Staubli VAL3: sampleChangerv5.pjx

--- sampleChangerv5.pjx ---
Parameters version=s7.7 stackSize=5000 millimeterUnit=true
Program file=comm.pgx
Program file=getNearestPos.pgx
Program file=getPosition.pgx
Program file=moveManager.pgx
Program file=observeStop.pgx
Program file=powerSwitch.pgx
Program file=sampleGripping.pgx
Program file=sendStatus.pgx
Program file=setSamPosOffs.pgx
Program file=setSpeed.pgx
Program file=setSpinPosOffs.pgx
Program file=start.pgx
Program file=stop.pgx
Program file=test.pgx
Program file=zsetSpinPosOffs.pgx
Data file=sampleChangerv5.dtx

--- sampleChangerV4.dtx ---
bool taskIsDone
dio switchGripper = {link=valve1}
jointRx binPosition = {j1=59.154914, j2=15.287075, j3=144.068937, j4=0.00349, j5=20.640131, j6=239.148927}
jointRx currentPickPosJ = {j1=24.086468, j2=103.725715, j3=36.339858, j4=-71.090092, j5=105.162663, j6=322.602811}
jointRx currentSamPosJ = {j1=64.5166, j2=21.7725, j3=135.395, j4=0.005, j5=22.8226, j6=244.506}
jointRx gatePosition = {j1=53.332436, j2=31.008098, j3=108.023775, j4=-0.035914, j5=40.963114, j6=323.353672}
jointRx homePosition = {j1=64.5166, j2=21.7725, j3=135.395, j4=0.005, j5=22.8226, j6=244.506}
jointRx parkingPosition = {j1=20.774519, j2=86.925335, j3=58.285959, j4=-72.455135, j5=101.349332, j6=295.989419}
jointRx spinnerPosition = {j1=24.224814, j2=103.543996, j3=36.557875, j4=-70.964584, j5=105.220885, j6=322.664695}
jointRx zeroPosition = {j1=88.745927, j2=-26.51301, j3=117.695598, j4=-0.539561, j5=89.308877, j6=269.442332}
mdesc mFastMov = {blend=off}
mdesc mNomSpeed = {accel=2.25, vel=15, decel=2.25}
num coords[2]
  [0] = 4
  [1] = 9
num numMessage[32]
num numSpeed = 5
num numXarray = 1
num numXold
num numYarray = 1
num numYold
pointRx currentPickPos = {x=982.652852, y=394.034002, z=-652.657917, rx=90.013165, ry=0.023145, rz=89.994895, shoulder=lefty, elbow=epositive, wrist=wpositive, fatherId=world[0]}
pointRx currentSamPos = {x=188.431145, y=511.898865, z=-95.729646, rx=-179.992666, ry=0.001448, rz=-0.004557, shoulder=lefty, elbow=epositive, wrist=wpositive, fatherId=world[0]}
sio sioASCII[2]
  [0] = {link=Socket\tan}
  [1] = {link=Socket\tan}

--- sampleChangerv5.dtx ---
bool moveIsStopped
dio switchGripper = {link=valve1}
jointRx binPosition = {j1=59.154914, j2=15.287075, j3=144.068937, j4=0.00349, j5=20.640131, j6=239.148927}
jointRx currentSamPosJ = {j1=64.5166, j2=21.7725, j3=135.395, j4=0.005, j5=22.8226, j6=244.506}
jointRx currentSpinPosJ
jointRx gatePosition = {j1=53.332436, j2=31.008098, j3=108.023775, j4=-0.035914, j5=40.963114, j6=323.353672}
jointRx homePosition = {j1=64.5166, j2=21.7725, j3=135.395, j4=0.005, j5=22.8226, j6=244.506}
jointRx knownPositions{}
  [currentSamPos] = {}
  [currentSpinPos] = {}
  [gatePosition] = {}
  [homePosition] = {}
  [parkingPosition] = {}
  [spinnerHomePos] = {}
  [zeroPosition] = {}
  [binPosition] = {}
jointRx parkingPosition = {j1=20.774519, j2=86.925335, j3=58.285959, j4=-72.455135, j5=101.349332, j6=295.989419}
jointRx spinnerHomePos = {j1=24.038951, j2=102.353577, j3=38.089715, j4=-71.031763, j5=105.005317, j6=322.961782}
jointRx zeroPosition = {j1=88.745927, j2=-26.51301, j3=117.695598, j4=-0.539561, j5=89.308877, j6=269.442332}
mdesc mFastMov = {blend=off}
mdesc mNomSpeed = {accel=2.25, vel=15, decel=2.25}
num numSamOffs[2]
num numSpinOffs[6]
sio sioASCII[2]
  [0] = {link=Socket\tan}
  [1] = {link=Socket\tan}
bool mounted
string calibInfo

--- start.pgx ---
program start()
begin
  call comm()
end

--- closeGripper.pgx ---
program closeGripper()
begin
  switchGripper=false
  taskKill("closeGripper")
end

--- comm.pgx ---
program comm()
  local num asciiMessage[64]
  local string command
  local string gripState
  local num nchars
  local string reply
  local num sio_ID
  local string stringMessage
  local num stringPos
  local bool waitForMessage
  local num msgLength
begin
  put("Starting sampleChangerV5.1...")
  //Disconnect running sessions
  clearBuffer(sioASCII)
  // We initialise the current sample position as the homePosition for safety's sake!
  currentSamPosJ=homePosition
  stringMessage=""
  reply=""
  msgLength=0

  // Populate the collection of known positions
  knownPositions["binPosition"] = binPosition
  knownPositions["currentSamPos"] = currentSamPosJ
  knownPositions["currentSpinPos"] = currentSpinPosJ
  knownPositions["gatePosition"] = gatePosition
  knownPositions["homePosition"] = homePosition
  knownPositions["parkingPosition"] = parkingPosition
  knownPositions["spinnerHomePos"] = spinnerHomePos
  knownPositions["zeroPosition"] = zeroPosition

  userPage()
  cls()

  putln("sampleChangerV5.1 server started.")
  putln("Waiting for command...")

  // Provides the server-like behaviour
  while true

    // The next while loop handles receiving messages.
    // The only way out is to recieve a message terminated with a ;
    waitForMessage=true
    while waitForMessage
      // The sioASCII socket allows two connections. We need to check which has something it it
      // Read recv buffer & place ASCII values in asciiMessage
      nchars=sioGet(sioASCII[0],asciiMessage)
      if nchars>0
        sio_ID=0
      else
        nchars=sioGet(sioASCII[1],asciiMessage)
        if nchars>0
          sio_ID=1
        else
        endIf
      endIf
      // Useful for debugging how many chars were received by the server
      //put("nchars: ")
      //putln(nchars)

      // sioGet returns a ASCII bytes. We need to decode them.
      if nchars>0
        stringMessage=chr(asciiMessage[0])
        for stringPos=1 to 63
          stringMessage=stringMessage+chr(asciiMessage[stringPos])
        endFor
        // We are finished with asciiMessage. Clear it
        for stringPos=0 to 63
          asciiMessage[stringPos]=0
        endFor

        // Check the last character in the message was a message end char (;)
        // If not, inform the sender and don't do anything
        if right(stringMessage,1)==";"
          stringMessage=left(stringMessage,len(stringMessage)-1)
          waitForMessage=false
        else
          call sendStatus(":fail_'No message end'",sio_ID)
          stringMessage=""
        endIf
        // Useful for debugging what was received by the server
        //put("stringMessage: ")
        //putln(stringMessage)
      endIf
    endWhile


    // All incoming messages should be of the form:
    //   command[:parameters]
    // Trim off the parameters for the switch statement
    stringPos=find(stringMessage,":")
    if stringPos>0
      command=left(stringMessage,stringPos)
    else
      command=stringMessage
    endIf
    put("Command: ")
    putln(command)

    //Now decide how to handle the message
    switch command
      // Testing routines
      // **********
      case "hello"
        call sendStatus("world",sio_ID)
      break

      case "test"
        call test()
      break

      // Control routines
      // **********
      case "setSamPosOffset"
        taskCreate "setSamPosOffset",10,setSamPosOffs(stringMessage,sio_ID)
        wait(taskStatus("setSamPosOffset")==-1)
      break

      case "getSamPosOffset"
        reply="getSamPosOffset:#X"+toString(".3",numSamOffs[0])
        reply=reply+"#Y"+toString(".3",numSamOffs[1])
        call sendStatus(reply,sio_ID)
      break

      case "setSpinPosOffset"
        taskCreate "setSpinPosOff",10,setSpinPosOffs(stringMessage,sio_ID)
        wait(taskStatus("setSpinPosOff")==-1)
      break

      case "getSpinPosOffset"
        reply="getSpinPosOffset:#X"+toString(".3",numSpinOffs[0])+"#Y"+toString(".3",numSpinOffs[1])
        reply=reply+"#Z"+toString(".3",numSpinOffs[2])+"#RX"+toString(".1",numSpinOffs[3])
        reply=reply+"#RY"+toString(".1",numSpinOffs[4])+"#RZ"+toString(".1",numSpinOffs[5])
        call sendStatus(reply,sio_ID)
      break

      case "getSpinPosition"
        call getPosition("getSpinPosition",currentSpinPosJ,sio_ID)
      break

      case "getSpinHomePosition"
        call getPosition("getSpinHomePosition",spinnerHomePos,sio_ID)
      break

      case "getCurrentPosition"
        call getPosition("getCurrentPosition",herej(),sio_ID)
      break

      case "getNearestPosition"
        call getNearestPos(sio_ID)
      break

      case "setCalibInfo"
        // Sets calibration info string
        msgLength = len(stringMessage)
        calibInfo = mid(stringMessage, (msgLength - 13), 13)
        call sendStatus("setCalibInfo:done", sio_ID)
      break

      case "getCalibInfo"
       reply = "getCalibInfo:" + calibInfo
       call sendStatus(reply,sio_ID)
      break

      case "setSpeed"
        taskCreate "setSpeed",5,setSpeed(stringMessage,sio_ID)
        wait(taskStatus("setSpeed")==-1)
      break

      case "getSpeed"
        call sendStatus("getSpeed:#"+toString("",mFastMov.vel),sio_ID)
      break

      case "powerOn"
        putln("Enabling robot power ...")
        taskCreate "powerSwitch",10,powerSwitch(true,"powerOn",sio_ID)
      break

      case "powerOff"
        putln("Disabling robot power ...")
        taskCreate "powerSwitch",10,powerSwitch(false,"powerOff",sio_ID)
      break

      case "getPowerState"
        putln("Get power status ...")
        if (isPowered()==false)
          reply="getPowerState:#Off"
        else
          reply="getPowerState:#On"
        endIf
        taskCreate "sendStatus",10,sendStatus(reply,sio_ID)
      break

      case "interrupt"
        putln("Interrupt movement ...")
        // Temporarily stops movement. This is basically a pause!\
        // Used by observeStop
        moveIsStopped=true
        call sendStatus("interrupt:done", sio_ID)
      break

      case "restart"
        putln("Restart from interruption ...")
        // Used by observeStop
        moveIsStopped=false
        call sendStatus("restart:done", sio_ID)
      break

      case "getGripperState"
        if switchGripper==true
          gripState="closed"
        else
          gripState="open"
        endIf
        call sendStatus("getGripperState:"+gripState,sio_ID)
      break

      // Movement routines
      // **********
      // Home position for the sample (sam)
      case "moveHome"
        putln("Moving to home ...")
        taskCreate "moveHome",10,moveManager(homePosition,mFastMov,"moveHome:done",sio_ID)
      break

      //Move to current sample offset position (home + offset)
      case "moveSamPos"
        putln("Moving to current sample ...")
        taskCreate "moveSamPos",10,moveManager(currentSamPosJ,mFastMov,"moveSamPos:done",sio_ID)
      break

      case "moveGate"
        putln("Moving to gate ...")
        taskCreate "moveGate",10,moveManager(gatePosition,mFastMov,"moveGate:done",sio_ID)
      break

      // Home position (calibrated) for the spinner
      case "moveSpinHome"
        putln("Moving to spinner home ...")
        taskCreate "moveSpinHome",10,moveManager(spinnerHomePos,mFastMov,"moveSpinHome:done",sio_ID)
      break

      //Move to current spinner offset position (spinnerHome + offset)
      case "moveSpinner"
        putln("Moving to spinner ...")
        taskCreate "moveSpinner",10,moveManager(currentSpinPosJ,mFastMov,"moveSpinner:done",sio_ID)
      break

      case "moveOffside"
        putln("Moving to offside ...")
        taskCreate "moveOffside",10,moveManager(parkingPosition,mFastMov,"moveOffside:done",sio_ID)
      break

      case "moveZero"
        putln("Moving to zero ...")
        taskCreate "moveZero",10,moveManager(zeroPosition,mFastMov,"moveZero:done",sio_ID)
      break

      case "moveBin"
        putln("Moving to bin ...")
        taskCreate "moveBin",10,moveManager(binPosition,mFastMov,"moveBin:done",sio_ID)
      break

      // Sample Handling
      // **********
      case "samplePick"
        putln("Picking sample ...")
        taskCreate "sampleGripping",10,sampleGripping(true,"samplePick",sio_ID)
      break

      case "sampleRelease"
        putln("Releasing sample ...")
        taskCreate "sampleGripping",10,sampleGripping(false,"sampleRelease",sio_ID)
      break

      case "gripperOpen"
        putln("Open gripper ...")
        switchGripper=false
        taskCreate "sendStatus",10,sendStatus("gripperOpen:done",sio_ID)
      break

      case "gripperClose"
        putln("Close gripper ...")
        switchGripper=true
        taskCreate "sendStatus",10,sendStatus("gripperClose:done",sio_ID)
      break

      case "isSampleMounted"
        // Check the state of the sample mounted flag
        if mounted == true
          reply = "isSampleMounted:#Yes"
        else
          reply = "isSampleMounted:#No"
        endIf
        call sendStatus(reply, sio_ID)
      break

      case "sampleMounted"
        // Set the sample mounted flag mounted (this is only s software flag)
        mounted = true
        taskCreate "sendStatus", 10, sendStatus("sampleMounted:done", sio_ID)
      break

      case "sampleUnmounted"
        // Set the sample mounted flag not mounted (this is only a software flag)
        mounted = false
        taskCreate "sendStatus", 10, sendStatus("sampleUnmounted:done", sio_ID)
      break

      default
        call sendStatus(":fail_'Unrecognised Command!'",sio_ID)
      break

    endSwitch
    // This message has been processed, so clear the stringMessage/command
    stringMessage=""
    command=""
    sio_ID=-1
    reply=""
    msgLength=0

  endWhile
end

--- getPosition.pgx ---
program getPosition(string getCommandName, joint requestedJoint, num sio_ID)
  local string message
  local pointRx readPosition
begin
  //**************************************************
  // Returns the contents of the trsf of the requested position.
  // On testing, we found that whereas a distance can be requested with
  // 2 or 3dp of precision, angles could not (got a runtime error on
  // the robot. Hence we return angles with no dp; we only need 2dp for
  // distances.
  //**************************************************
  putln("getPosition:")
  putln("   "+getCommandName)
  readPosition=jointToPoint(flange,world,requestedJoint)
  message=getCommandName+":#X"+toString(".2",readPosition.trsf.x)
  message=message+"#Y"+toString(".2",readPosition.trsf.y)
  message=message+"#Z"+toString(".2",readPosition.trsf.z)
  message=message+"#RX"+toString("",readPosition.trsf.rx)
  message=message+"#RY"+toString("",readPosition.trsf.ry)
  message=message+"#RZ"+toString("",readPosition.trsf.rz)

  call sendStatus(message,sio_ID)
end

--- moveBin.pgx ---
program moveBin()
begin
  movej(binPosition,flange,mFastMov)
  waitEndMove()
  message="moveBin:done"
  taskCreate "sendStatus",10,sendStatus()
  taskKill("moveBin")
end

--- moveGate.pgx ---
program moveGate()
begin
  movej(gatePosition,flange,mFastMov)
  waitEndMove()
  message="moveGate:done"
  taskCreate "sendStatus",100,sendStatus()
  taskKill("moveGate")
end

--- moveHome.pgx ---
program moveHome()
begin
  movej(homePosition,flange,mFastMov)
  waitEndMove()
  message="moveHome:done"
  taskCreate "sendStatus",100,sendStatus()
  taskKill("moveHome")
end

--- moveManager.pgx ---
program moveManager(joint destination (dimensions=1), mdesc armSpeed (dimensions=1), string reply (dimensions=1), num sio_ID (dimensions=1))
begin
  //**************************************************
  // Method to enable joint-based movements of the robot. The referenced
  // observeStop() method allows interrupts/restarts to be handled
  //**************************************************
  taskIsDone=false
  taskCreate "observeStop",5,observeStop()
  movej(destination,flange,armSpeed)
  waitEndMove()
  taskCreate "sendStatus",10,sendStatus(reply,sio_ID)
  taskKill("observeStop")
end

--- moveNext.pgx ---
program moveNext()
begin
  currentSamPosJ=herej()
  currentSamPos=jointToPoint(flange,world,currentSamPosJ)
  movel(appro(currentSamPos,{(numXarray-1)*-17.03,(numYarray-1)*-17,0,0,0,0}),flange,mFastMov)
  waitEndMove()
end

--- moveOffside.pgx ---
program moveOffside()
begin
  movej(parkingPosition,flange,mFastMov)
  waitEndMove()
  message="moveOffside:done"
  taskCreate "sendStatus",100,sendStatus()
  taskKill("moveOffside")
end

--- moveSpinner.pgx ---
program moveSpinner()
begin
  movej(spinnerPosition,flange,mFastMov)
  waitEndMove()
  message="moveSpinner:done"
  taskCreate "sendStatus",100,sendStatus()
  taskKill("moveSpinner")
end

--- moveZero.pgx ---
program moveZero()
begin
  movej(zeroPosition,flange,mFastMov)
  waitEndMove()
  message="moveZero:done"
  taskCreate "sendStatus",100,sendStatus()
  taskKill("moveZero")
end

--- notGrip.pgx ---
program notGrip()
begin
  if switchGripper==true
    switchGripper=false
  else
  endIf
end

--- observeStop.pgx ---
program observeStop()
begin
  //**************************************************
  // Method interrupts a running move operation. This is
  // equivalent to a pause.
  //
  // Method is triggered by a flag being set.
  // N.B. Move is only stopped until flag is unset.
  //**************************************************
  while true
    wait(moveIsStopped==true)
    stopMove()
    wait(moveIsStopped==false)
    restartMove()
  endWhile
end

--- openGripper.pgx ---
program openGripper()
begin
  switchGripper=false
  message="openGripper:done"
  taskCreate "sendStatus",100,sendStatus()
  taskKill("openGripper")
end

--- pickSample.pgx ---
program pickSample()
begin
  taskCreate "notGrip",100,notGrip()
  currentSamPosJ=herej()
  currentSamPos=jointToPoint(flange,world,currentSamPosJ)
  movel(appro(currentSamPos,{0,0,80,0,0,0}),flange,mNomSpeed)
  waitEndMove()
  taskKill("notGrip")
  switchGripper=true
  movel(appro(currentSamPos,{0,0,0,0,0,0}),flange,mNomSpeed)
  waitEndMove()
  message="pickSample:done"
  taskCreate "sendStatus",100,sendStatus()
  taskKill("pickSample")
  //taskKill("notGrip")
end

--- powerOff.pgx ---
program powerOff()
begin
  disablePower()
  message="disablePower:done"
  taskCreate "sendStatus",100,sendStatus()
  taskKill ("powerOff")
end

--- powerOn.pgx ---
program powerOn()
begin
 enablePower()
 if (watch(isPowered(),5)==false)
  putln("Arm power supply cannot be switched on")
 endIf
 message="enablePower:done"
 taskCreate "sendStatus",100,sendStatus()
 taskKill ("powerOn")
end

--- powerSwitch.pgx ---
program powerSwitch(bool enable (dimensions=1), string command (dimensions=1), num sio_ID (dimensions=1))
  local string reply
begin
  //**************************************************
  // Method to enable or disable the power on the robot, depending whether the
  // enable variable is true or false. Command argument is needed to construct
  // the reply
  //**************************************************
  if enable
    enablePower()
  else
    disablePower()
  endIf

  if (watch(isPowered()==enable,5)==false)
    reply=command+":fail_'RobotPowerCannotBeSwitched'"
  else
    reply=command+":done"
  endIf
  taskCreate "sendStatus",10,sendStatus(reply,sio_ID)
  taskKill("powerSwitch")
end

--- releaseSample.pgx ---
program releaseSample()
begin
  currentSamPosJ=herej()
  currentSamPos=jointToPoint(flange,world,currentSamPosJ)
  movel(appro(currentSamPos,{0,0,80,0,0,0}),flange,mNomSpeed)
  waitEndMove()
  switchGripper=false
  movel(appro(currentSamPos,{0,0,0,0,0,0}),flange,mNomSpeed)
  waitEndMove()
  message="releaseSample:done"
  taskCreate "sendStatus",100,sendStatus()
  taskKill ("releaseSample")
end

--- reset.pgx ---
program reset()
begin
  //putln(taskStatus("closeGripper"))
  if taskStatus("closeGripper")==1
    taskKill("closeGripper")
  endIf
  if taskStatus("moveBin")==1
    taskKill("moveBin")
  endIf
  if taskStatus("moveGate")==1
    taskKill("moveGate")
  endIf
  if taskStatus("moveHome")==1
    taskKill("moveHome")
  endIf
  if taskStatus("moveOffside")==1
    taskKill("moveOffside")
  endIf
  if taskStatus("moveZero")==1
    taskKill("moveZero")
  endIf
  if taskStatus("pickSample")==1
    taskKill("pickSample")
  endIf
  if taskStatus("releaseSample")==1
    taskKill("releaseSample")
  endIf
  if taskStatus("stopMotor")==1
    taskKill("stopMotor")
  endIf
  if taskStatus("restartMotor")==1
    taskKill("restartMotor")
  endIf
  stopMove()
  resetMotion()
end

--- restartMotor.pgx ---
program restartMotor()
begin
  restartMove()
  message="restartMove:done"
  taskCreate "sendStatus",100,sendStatus()
  taskKill ("restartMotor")
end

--- sampleGripping.pgx ---
program sampleGripping(bool gripSample (dimensions=1), string command (dimensions=1), num sio_ID (dimensions=1))
  local jointRx pickingPosJoint
  local pointRx pickingPosPoint
  local string reply
begin
  //**************************************************
  // Method to take or place sample at the magazine or at the spinner.
  // The former is determined by the gripSample argument. The latter
  // is determined from the position (herej()) of the arm when this
  // method is called.
  //**************************************************

  // For picking samples (we end with sample in the gripper), we must have an open
  // gripper to start with
  if (gripSample==true) and (switchGripper==true)
    switchGripper=false
  else
  endIf

  // The current pick position is either the currentSamPosJ or spinnerPosition
  // We don't know which and to make this flexible we set for the scope of this method
  pickingPosJoint=herej()
  pickingPosPoint=jointToPoint(flange,world,pickingPosJoint)
  // Move in to the sample
  movel(appro(pickingPosPoint,{0,0,80,0,0,0}),flange,mNomSpeed)
  waitEndMove()

  // Grab the sample and move out
  switchGripper=gripSample
  movel(appro(pickingPosPoint,{0,0,0,0,0,0}),flange,mNomSpeed)
  waitEndMove()

  reply=command+":done"
  taskCreate "sendStatus",10,sendStatus(reply,sio_ID)
  taskKill("sampleGripping")

end

--- sendStatus.pgx ---
program sendStatus()
begin
  for stringLen=0 to 15
    message2ASCII[stringLen]=asc(mid(message,1,stringLen),0)
  endFor
  sioSet(sioASCII,message2ASCII)
  delay(1)
end

--- setCoords.pgx ---
program setCoords(string inputMessage (dimensions=1), num sio_ID (dimensions=1))
  local bool isNumber[2]
  local bool isOK
  local num msgLength
  local string reply
  local pointRx sampleCoordPnt
  local num xMsgIndex
  local num yMsgIndex
begin
  //**************************************************
  // Method to set the coordinates of currentSamPosj (current sample position).
  // Messages take the form:
  //     setCoords:#X1#Y2
  // Coordinate system starts at 0 (e.g. X=0, Y=0 is first sample position)
  //**************************************************

  // To start with the function is assumed working and we print the input
  isOK=true
  putln("Setting magazine coordinates based on:")
  putln("   "+inputMessage)


  // Find the where the coordinates are being supplied
  xMsgIndex=find(inputMessage,"#X")
  yMsgIndex=find(inputMessage,"#Y")
  msgLength=len(inputMessage)

  // Extract the coords from the message and convert string to number
  toNum(mid(inputMessage,(yMsgIndex-(xMsgIndex+2)),(xMsgIndex+2)),coords[0],isNumber[0])
  toNum(mid(inputMessage,(msgLength-(yMsgIndex+2)),(yMsgIndex+2)),coords[1],isNumber[1])

  // Check conversion to number successful and print to screen
  isOK=isOK and isNumber[0] and isNumber[1]
  if isNumber[0]==false
    reply="setCoords:fail_'Invalid X'"
    put("Failed setting X. Found: ")
    putln(right(inputMessage,(yMsgIndex-(xMsgIndex+2))))
  elseIf isNumber[1]==false
    reply="setCoords:fail_'Invalid Y'"
    put("Failed setting Y. Found: ")
    putln(right(inputMessage,(msgLength-(yMsgIndex+2))))
  endIf

  // Assuming we got the numbers, now we create our new joint coordinate
  if isOK==true
    put("Coords: X=")
    put(coords[0])
    put(" Y=")
    putln(coords[1])
    sampleCoordPnt=appro(jointToPoint(flange,world,homePosition),{(coords[0])*-17.03,(coords[1])*-17,0,0,0,0})
    isOK=pointToJoint(flange,homePosition,sampleCoordPnt,currentSamPosJ)

    if isOK==false
      reply="setCoords:fail_'Could not convert position to joint'"
      putln("Failed converting position to joint")
    else
      reply="setCoords:done"
    endIf
  endIf

  taskCreate "sendStatus",10,sendStatus(reply,sio_ID)
  taskKill("setCoords")
end

--- setSAM.pgx ---
program setSAM(string messageBuffer (dimensions=1), string message (dimensions=1), num sio_ID (dimensions=1))
  local num indexX
  local num indexY
  local num indexZ
  local bool isnum
  local num samX
  local num samY
  local num samZ
begin
  putln(messageBuffer)
  currentPickPosJ=herej()
  currentPickPos=jointToPoint(flange,world,currentPickPosJ)
  //numXold=numXarray
  //numYold=numYarray
  indexX=find(messageBuffer,("#Y"))
  indexZ=find(messageBuffer,("#Z"))
  toNum(left(messageBuffer,indexX),samX,isnum)
  if isnum==false
    taskCreate "sendStatus",10,sendStatus("... X is not a number ...",sio_ID)
    putln("... X is not a number ...")
  endIf
  indexY=len(messageBuffer)-find(messageBuffer,("#Z"))-2
  toNum(right(messageBuffer,indexY),samY,isnum)
  if isnum==false
    taskCreate "sendStatus",10,sendStatus("... Y is not a number ...",sio_ID)
    putln("... Y is not a number ...")
  endIf
  toNum(mid(messageBuffer,indexZ-indexY,indexY+2),samZ,isnum)
  if isnum==false
    taskCreate "sendStatus",10,sendStatus("... Z is not a number ...",sio_ID)
    putln("... Z is not a number ...")
  endIf
  putln("show sam values:")
  putln(toString(".3",samX))
  putln(toString(".3",samY))
  putln(toString(".3",samZ))
  movel(appro(currentPickPos,{samY,-samX,-samZ,0,0,0}),flange,mNomSpeed)
  waitEndMove()
  taskCreate "sendStatus",10,sendStatus(message,sio_ID)
  putln(message)
  //required shape: e.g. 'setSAM#X1.12345#Y2.3456#Z0.2345'
end

--- setSamPosOffs.pgx ---
program setSamPosOffs(string inputMessage, num sio_ID)
  local bool isNumber[2]
  local bool isOK
  local num msgLength
  local string reply
  local pointRx samplePosPnt
  local num xMsgIndex
  local num yMsgIndex
begin
  //**************************************************
  // Method to set the coordinates of currentSamPosj (current sample position).
  // Messages take the form:
  //     setSamPosOffset:#X1#Y2
  // Coordinate system starts at 0 (e.g. X=0, Y=0 is first sample position)
  //**************************************************

  // To start with the function is assumed working and we print the input
  isOK=true
  putln("Setting magazine coordinates:")
  putln("   "+inputMessage)

  // Find the where the coordinates are being supplied
  xMsgIndex=find(inputMessage,"#X")
  yMsgIndex=find(inputMessage,"#Y")
  msgLength=len(inputMessage)

  // Extract the numSamPos from the message and convert string to number
  toNum(mid(inputMessage,(yMsgIndex-(xMsgIndex+2)),(xMsgIndex+2)),numSamOffs[0],isNumber[0])
  toNum(mid(inputMessage,(msgLength-(yMsgIndex+2)),(yMsgIndex+2)),numSamOffs[1],isNumber[1])

  // Check conversion to number successful and print to screen
  isOK=isOK and isNumber[0] and isNumber[1]
  if isNumber[0]==false
    reply="setSamPos:fail_'Invalid X'"
    put("Failed setting X. Found: ")
    putln(right(inputMessage,(yMsgIndex-(xMsgIndex+2))))
  elseIf isNumber[1]==false
    reply="setSamPos:fail_'Invalid Y'"
    put("Failed setting Y. Found: ")
    putln(right(inputMessage,(msgLength-(yMsgIndex+2))))
  endIf

  // Assuming we got the numbers, now we create our new joint coordinate
  if isOK==true
    put("SamPos: X=")
    put(numSamOffs[0])
    put(" Y=")
    putln(numSamOffs[1])
    samplePosPnt=appro(jointToPoint(flange,world,homePosition),{(numSamOffs[0])*-17.03,(numSamOffs[1])*-17,0,0,0,0})
    isOK=pointToJoint(flange,homePosition,samplePosPnt,currentSamPosJ)

    // Update knownPositions collection
    knownPositions["currentSamPos"] = currentSamPosJ

    if isOK==true
      reply="setSamPosOffset:done"
    else
      reply="setSamPosOffset:fail_'Could not convert position to joint'"
      putln("Failed converting position to joint")
    endIf
  endIf

  taskCreate "sendStatus",10,sendStatus(reply,sio_ID)
  taskKill("setSamPosOffset")
end

--- setSpeed.pgx ---
program setSpeed(string messageBuffer (dimensions=1), num sio_ID (dimensions=1))
  local num indexParam
  local bool isNumber
  local num numSpeedLoc
  local string reply
begin
  //**************************************************
  // Method to set the speed of the robot. Messages take the form:
  //     setSpeed:#20
  //**************************************************

  // Find the parameter in the stringMessage and convert to a number
  indexParam=find(messageBuffer,("#"))
  toNum(right(messageBuffer,(len(messageBuffer)-(indexParam+1))),numSpeedLoc,isNumber)

  // If conversion worked, set the speed; if not post a message and return
  if isNumber==false
    reply="setSpeed:fail_'Data is not a number'"
    putln(toString("",indexParam))
    putln(toString("",len(messageBuffer)-(indexParam+1)))
    put("Failed setting speed. Found: ")
    putln(right(messageBuffer,(len(messageBuffer)-indexParam)))
  else
    mFastMov.vel=numSpeedLoc
    put("Speed = ")
    putln(numSpeedLoc)
    reply="setSpeed:done"
  endIf

  taskCreate "sendStatus",10,sendStatus(reply,sio_ID)
end

--- setXaxis.pgx ---
program setXaxis()
begin
  numMessage[4]=0
  stringXarray=""
  while numMessage[4]==0
    sioGet(sioASCII,numMessage)
    stringXarray=chr(numMessage[0])
    if chr(numMessage[1])!="#"
      stringXarray=stringXarray+chr(numMessage[1])
    endIf
    toNum(stringXarray,numXarray,isNum)
    putln(stringXarray)
  endWhile
end

--- setYaxis.pgx ---
program setYaxis()
begin
  numMessage[4]=0
  //-------------------------------set carrier to default
  stringYarray=""
  while numMessage[4]==0
    sioGet(sioASCII,numMessage)
    stringYarray=chr(numMessage[0])
    if chr(numMessage[1])!="#"
      stringYarray=stringYarray+chr(numMessage[1])
      //stringYarray=chr(numMessage[4])
    endIf
    toNum(stringYarray,numYarray,isNum)
    putln(stringYarray)
  endWhile
end

--- stopMotor.pgx ---
program stopMotor()
begin
  stopMove()
  message="stopMotor:done"
  taskCreate "sendStatus",100,sendStatus()
  taskKill ("stopMotor")
end

--- zsetSpinPosOffs.pgx ---
program zsetSpinPosOffs(string inputMessage (dimensions=1), num sio_ID (dimensions=1))
  local bool isNumber[6]
  local bool isOK
  local num msgLength
  local string reply
  local num rxMsgIndex
  local num ryMsgIndex
  local num rzMsgIndex
  local pointRx spinnerPosPnt
  local num xMsgIndex
  local num yMsgIndex
  local num zMsgIndex
begin
  //**************************************************
  //
  // THIS VERSION IS AN EXAMPLE OF HOW TO DO ROTATIONS TOO
  // IT IS NOT NEEDED (as of 16.02.2020). IT IS NOT USED!!!!
  //
  //
  // Method to set the coordinates of currentSpinPosj (current spinner position).
  // Messages take the form:
  //     setSpinPos:#X1#Y2#Z3#RX4#RY5#RZ6
  // Coordinate system starts at robot world frame origin (e.g. X=0, Y=0, Z=0, rx=0, ry=0, rz=0)
  //**************************************************

  // To start with the function is assumed working and we print the input
  isOK=true
  putln("Setting spinner coordinates based on:")
  putln("   "+inputMessage)


  // Find the where the coordinates are being supplied
  xMsgIndex=find(inputMessage,"#X")
  yMsgIndex=find(inputMessage,"#Y")
  zMsgIndex=find(inputMessage,"#Z")
  //rxMsgIndex = find(inputMessage,"#RX")
  //ryMsgIndex = find(inputMessage,"#RY")
  //rzMsgIndex = find(inputMessage,"#RZ")
  msgLength=len(inputMessage)

  // Extract the numSpinPos from the message and convert string to number
  toNum(mid(inputMessage,(yMsgIndex-(xMsgIndex+2)),(xMsgIndex+2)),numSpinOffs[0],isNumber[0])
  toNum(mid(inputMessage,(zMsgIndex-(yMsgIndex+2)),(yMsgIndex+2)),numSpinOffs[1],isNumber[1])
  //  toNum(mid(inputMessage, (rxMsgIndex - (zMsgIndex + 2)), (zMsgIndex + 2)), numSpinOffs[2], isNumber[2])
  //  toNum(mid(inputMessage, (ryMsgIndex - (rxMsgIndex + 2)), (rxMsgIndex + 2)), numSpinOffs[3], isNumber[3])
  //  toNum(mid(inputMessage, (rzMsgIndex - (ryMsgIndex + 2)), (ryMsgIndex + 2)), numSpinOffs[4], isNumber[4])
  //  toNum(mid(inputMessage, (msgLength - (rzMsgIndex + 2)), (rzMsgIndex + 2)), numSpinOffs[5], isNumber[5])
  toNum(mid(inputMessage,(msgLength-(zMsgIndex+2)),(zMsgIndex+2)),numSpinOffs[2],isNumber[2])

  //  toNum(mid(inputMessage, (msgLength - (yMsgIndex + 2)), (yMsgIndex + 2)), numSamOffs[1], isNumber[1])

  // Check conversion to number successful and print to screen
  isOK=isOK and isNumber[0] and isNumber[1] and isNumber[2]
  //and isNumber[3] and isNumber[4] and isNumber[5]
  if isNumber[0]==false
    reply="setSpinPosOffset:fail_'Invalid X'"
    put("Failed setting X. Found: ")
    putln(right(inputMessage,(yMsgIndex-(xMsgIndex+2))))
  elseIf isNumber[1]==false
    reply="setSpinPosOffset:fail_'Invalid Y'"
    put("Failed setting Y. Found: ")
    putln(right(inputMessage,(zMsgIndex-(yMsgIndex+2))))
  elseIf isNumber[2]==false
    reply="setSpinPosOffset:fail_'Invalid Z'"
    put("Failed setting Z. Found: ")
    putln(right(inputMessage,(rxMsgIndex-(zMsgIndex+2))))
    //  elseIf isNumber[3] == false
    //    reply = "setSpinPosOffset:fail_'Invalid RX'"
    //    put("Failed setting RX. Found: ")
    //    putln(right(inputMessage, (ryMsgIndex - (rxMsgIndex + 2))))
    //  elseIf isNumber[4] == false
    //    reply = "setSpinPosOffset:fail_'Invalid RY'"
    //    put("Failed setting RY. Found: ")
    //    putln(right(inputMessage, (rzMsgIndex - (ryMsgIndex + 2))))
    //  elseIf isNumber[5] == false
    //    reply = "setSpinPosOffset:fail_'Invalid RZ'"
    //    put("Failed setting RZ. Found: ")
    //    putln(right(inputMessage, (msgLength - (rzMsgIndex + 2))))
  endIf

  // Assuming we got the numbers, now we create our new joint coordinate
  if isOK==true
    put("SpinPos: X=")
    put(numSpinOffs[0])
    put(" Y=")
    putln(numSpinOffs[1])
    put(" Z=")
    putln(numSpinOffs[2])
    //    put(" RX=")
    //    putln(numSpinOffs[3])
    //    put(" RY=")
    //    putln(numSpinOffs[4])
    //    put(" RY=")
    //    putln(numSpinOffs[5])
    spinnerPosPnt=compose(jointToPoint(flange,world,spinnerHomePos),world,{numSpinOffs[0],numSpinOffs[1],numSpinOffs[2],0,0,0})
    //  Don't use appro - it applies the current rx,ry,rz rotation to any translations requested
    //    spinnerPosPnt = appro(jointToPoint(flange,world,spinnerHomePos),{numSpinOffs[0],numSpinOffs[1],numSpinOffs[2],numSpinOffs[3],numSpinOffs[4],numSpinOffs[5]})
    //    spinnerPosPnt = appro(jointToPoint(flange,world,spinnerHomePos),{numSpinOffs[0],numSpinOffs[1],numSpinOffs[2],0,0,0})
    //
    //  The following would make the set absolute positions. It's better to use a fixed position (SpinnerHome) and apply offsets
    //    currentPickPos.trsf.x = numSpinOffs[0]
    //    currentPickPos.trsf.y = numSpinOffs[1]
    //    currentPickPos.trsf.z = numSpinOffs[2]
    //    currentPickPos.trsf.rx = numSpinOffs[3]
    //    currentPickPos.trsf.ry = numSpinOffs[4]
    //    currentPickPos.trsf.rz = numSpinOffs[5]
    isOK=pointToJoint(flange,spinnerHomePos,spinnerPosPnt,currentSpinPosJ)
    // We are using a joint arrangement in spinnerPosition from before v5 because it worked!

    if isOK==true
      reply="setSpinPosOffset:done"
    else
      reply="setSpinPosOffset:fail_'Could not convert position to joint'"
      putln("Failed converting position to joint")
    endIf
  else
    reply="setSpinPosOffset:fail_'Offset setting failed for unknown reason'"
    putln("Failed setting offset: reason unknown'")
  endIf

  taskCreate "sendStatus",10,sendStatus(reply,sio_ID)
  taskKill("setSpinPosOff")
end
